PROGRAM MAIN
VAR
	//Devices
	EL3443_Terminal			: MDP5001_341_A3044239;
	fbspeedwire				: FB_SPEEDWIRE;
END_VAR

fbspeedwire(
	EL3443 := EL3443_Terminal
	);

END_PROGRAM

(* stored: Version 1.1.0.1, ProductVersion 3.1.4024.12
   POU MAIN: Id {3fc796c7-da3a-491a-9e37-cc741c45d921}, SpecialFunc None *)
